SUBAPPLICATION SubApp_PC_B (* Geraet B (Station 12, 192.168.1.12): Toggle-Flipflop-Logik (AE_AX_T_FF) und DigitalOutput_Q1 - 'SUB style', das Protokoll steckt im MyLib::sys-Composite (SoftKeyT_PC_B_OPC_Adapter), nicht in der Resource des Geraets - Adapter-Variante von Training_08, gleiche OPC-UA-Adressen wie Training_03 *)
  (* Standard: 61499-2; Description: Copyright (c) 2026 Meisterschulen am Ostbahnhof This program and the accompanying materials are made available under the terms of the Eclipse Public License 2.0 which is available at https://www.eclipse.org/legal/epl-2.0/ SPDX-License-Identifier: EPL-2.0 *)
  (* Version 1.0, 2026-09-04, Franz Höpfinger, Meisterschulen am Ostbahnhof, initial API and implementation and/or initial documentation *)
  PACKAGE subapp::Training_09_OPC_UA_RES;
  IMPORT logiBUS::io::DQ::logiBUS_DO::Output_Q1;
  IMPORT VV::const::OPC_UA::myOpcUaAddresses::FF1_TRIGGER_LOCAL_METHOD;
  IMPORT VV::const::OPC_UA::myOpcUaAddresses::FF1_STATE_REMOTE_WRITE;
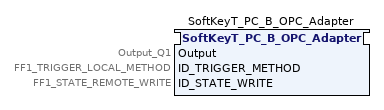
  SUBAPPS
    SoftKeyT_PC_B_OPC_Adapter : MyLib::sys::SoftKeyT_PC_B_OPC_Adapter(Output := Output_Q1, ID_TRIGGER_METHOD := FF1_TRIGGER_LOCAL_METHOD, ID_STATE_WRITE := FF1_STATE_REMOTE_WRITE);
  END_SUBAPPS
END_SUBAPPLICATION
